FUNCTION_BLOCK ByteBufferFileWriter
VAR
	state : (IDLE, OPEN, OPENING, OPENED, WRITE, WRITING, WRITTEN, CLOSE, CLOSING, CLOSED, ERROR) := IDLE;
	netId : T_AmsNetId := '';	
	fileName : T_MaxString := '';
	errId : UDINT;
	hFile : UINT := 0;
	byteBuffer : I_Buffer;
	fbFileOpen : FB_FileOpen;
	fbFileClose : FB_FileClose;
	fbFileWrite : FB_FileWrite;
END_VAR

CASE state OF
	IDLE: //

	OPEN:
	
		errId := 0;
		fbFileOpen(bExecute := FALSE);
		fbFileOpen( 
			sNetId := netId, 
			sPathName := fileName, 
			nMode := FOPEN_MODEWRITE OR FOPEN_MODEBINARY, 
			ePath := PATH_GENERIC, 
			bExecute := TRUE 
		);
			
		state := OPENING;

	OPENING:
	
		fbFileOpen( 
			bExecute := FALSE,
			hFile => hFile 
		);
		
		IF NOT fbFileOpen.bBusy THEN
			IF NOT fbFileOpen.bError THEN
				state := OPENED;
			ELSE
				state := ERROR;
				errId := fbFileOpen.nErrId;
			END_IF
		END_IF

	OPENED: //

	WRITE:	
	
		fbFileWrite(bExecute := FALSE );
		fbFileWrite( 
			sNetId := netId, 
			hFile := hFile, 
			pWriteBuff := byteBuffer.Address, 
			cbWriteLen := byteBuffer.Size, 
			bExecute := TRUE 
		);
		state := WRITING;

	WRITING:

		fbFileWrite( 
			bExecute := FALSE
		);
		
		IF NOT fbFileWrite.bBusy THEN
			IF NOT fbFileWrite.bError THEN
				state := WRITTEN;
			ELSE
				state := ERROR;
				errId := fbFileWrite.nErrId;
			END_IF
		END_IF

	WRITTEN: state := OPENED;
	
	CLOSE:	
	
		fbFileClose(bExecute := FALSE);
		fbFileClose( 
			sNetId := netId, 
			hFile := hFile, 
			bExecute := TRUE 
		);
		state := CLOSING;

	CLOSING:
	
		fbFileClose( 
			bExecute := FALSE
		);
		
		IF ( NOT fbFileClose.bBusy ) THEN
			hFile := 0;
			state := CLOSED;
		END_IF

	CLOSED: state := IDLE;
	
	ERROR:
		
		IF ( hFile <> 0 ) THEN
			state := CLOSE; 
		ELSE
			state := IDLE;
		END_IF

END_CASE

METHOD PUBLIC CloseFile : BOOL
IF state = OPENED THEN
	state := CLOSE;
	CloseFile := TRUE;
END_IF
END_METHOD

METHOD FB_init : BOOL
VAR_INPUT
	bInitRetains : BOOL; // if TRUE, the retain variables are initialized (warm start / cold start)
	bInCopyCode : BOOL;  // if TRUE, the instance afterwards gets moved into the copy code (online change)
	NetId : T_AmsNetId; // Leave blank for local
END_VAR
this^.netId := NetId;
END_METHOD

PROPERTY PUBLIC IsBusy : BOOL
GET
IsBusy := NOT (state = IDLE OR state = OPENED);
END_GET
END_PROPERTY

PROPERTY PUBLIC IsClosed : BOOL
GET
IsClosed := (state = IDLE);
END_GET
END_PROPERTY

PROPERTY PUBLIC IsOpen : BOOL
GET
IsOpen := not IsClosed and not (state = OPENING or state = OPEN);
END_GET
END_PROPERTY

METHOD PUBLIC OpenFile : BOOL
VAR_INPUT
	FileName : T_MaxString;
END_VAR
IF FileName = '' THEN
	RETURN;
END_IF

IF state = IDLE THEN
	THIS^.fileName := FileName;
	state := OPEN;
	OpenFile := TRUE;
END_IF
END_METHOD

METHOD PUBLIC WriteByteBufferToFile : BOOL
VAR_INPUT
	buffer : I_Buffer;
END_VAR
IF buffer = 0 THEN
	RETURN;
END_IF

IF buffer.Size = 0 THEN
	RETURN;
END_IF

IF state = OPENED THEN
	THIS^.byteBuffer := buffer;
	state := WRITE;
	WriteByteBufferToFile := TRUE;
END_IF
END_METHOD

PROPERTY PUBLIC WriteComplete : BOOL
GET
WriteComplete := state = WRITTEN;
END_GET
END_PROPERTY

END_FUNCTION_BLOCK

(* stored: Version 1.1.0.1, ProductVersion 3.1.4024.4
   POU ByteBufferFileWriter: Id {974330a0-7c08-4b2f-b77a-a168cef059fe}, SpecialFunc None
   Method CloseFile: Id {1e9eada9-7a1e-48f9-a23e-4ca727eb0055}
   Method FB_init: Id {d86f9bb2-8e65-4992-832b-c69498cbf4bf}
   Property IsBusy: Id {adf99bea-4af0-48c3-88aa-39b232ec5c96}
   Get Get: Id {bdbeb253-5353-46af-be39-7f4024c85203}
   Property IsClosed: Id {53110810-2495-4881-9bd3-64111837d44a}
   Get Get: Id {c9f4dd2f-ba5c-4d7b-8562-cfdd8ad65252}
   Property IsOpen: Id {b162d915-0c49-4a6e-8da9-aa6208295a34}
   Get Get: Id {fbeae986-de40-45e8-aa23-da8880829ab0}
   Method OpenFile: Id {d656c749-7bb1-4d56-ab15-9a5e6a25769b}
   Method WriteByteBufferToFile: Id {b1b948ae-968f-414b-b01d-51099a4dd98f}
   Property WriteComplete: Id {c19a5449-807d-44cb-87c1-322474441acc}
   Get Get: Id {0053eaca-b4ff-4762-b1c1-8d788f325f46} *)
